(* Logix 5000 project; controller PRU vendor 1 type 14 code 107 rev 20.13; software revision 20.01; part 5 of 17 *)
(* tags used below, declared in another part *)
   AFI : BOOL;
   AlarmMaster : DINT;
   ALL_AUTO_IOK : BOOL;   // All equipment is in Auto Mode.
   ALL_DRIVES_ARE_CMD_FWD : BOOL;
   ALL_DRIVES_ARE_READY : BOOL;
   ALL_SHUTDOWN_FAULTS_IOK : BOOL;
   AUTO_DISCHARGE_CYCLE_ION : BOOL;   // Proces Sequencer (4-13)
   AUTO_SHUTDOWN_ENABLE : BOOL;
   CLEARING_PYROLIZER_TIME_REMAINING_SEC : REAL;
   CLEARING_PYROLIZER_TIME_REMAINING_TEMP : REAL;
   CLEARING_PYROLIZER_TIMER : TIMER;
   COOLSCREW : VFD;
   CR0_CON1_HTR1_GON : BOOL;   // ZONE 1 (L1,L2,L3)
   CR1_CON2_HTR2_GON : BOOL;   // ZONE 2 (L1,L2,L3)
   CR2_CON3_HTR3_GON : BOOL;   // ZONE 3 (L1,L2,L3)
   CR3_CON4_HTR4_GON : BOOL;   // ZONE 4 (L1) ZONE 5 (L2) ZONE 6 (L3)
   CR4_CON5_HTR5_GON : BOOL;   // ZONE 7 (L1) ZONE 8 (L2) ZONE 9 (L3)
   DRYER_MODE_AUTO : BOOL;
   FAULTS_FA1_IOK : BOOL;   // SYSTEM LEVEL FAULTS ARE OK.
   FAULTS_FA3A_IOK : BOOL;   // SCREWS DRIVES NOT FAULTED.
   FAULTS_FA3B_IOK : BOOL;   // ENCODERS NOT FAULTED.
   FAULTS_FA4_IOK : BOOL;   // HI TEMP FAULTS ARE OK.
   FAULTS_FA5_IOK : BOOL;
   FAULTS_FA5A_IOK : BOOL;   // COOLING SCREW FAULTS ARE OK.
   FAULTS_FA5C_IOK : BOOL;   // KG021 FAULTS ARE OK.
   FAULTS_FA5D_IOK : BOOL;   // KG021 FAULTS ARE OK.
   FAULTS_FA6_IOK : BOOL;   // HEATER FAULTS ARE OK.
   FINISH_PROCESS_TIME_REMAINING_SEC : REAL;
   FINISH_PROCESS_TIME_REMAINING_TEMP : REAL;
   FINISH_PROCESS_TIMER : TIMER;
   FS0101_ION : BOOL;   // LOW FLOW SWITCH - INLET AND DISCHARGE PURGE
   HEATER_FAULTS_IOK : BOOL;   // FA1, FA4, FA6
   HEATERS_CYCLE_ION : BOOL;   // Heaters are commanded on.
   HMI_ABORT_PB : BOOL;
   HMI_AUTO_START_PB : BOOL;
   HMI_CLEARING_PYROLIZER_TIME_MIN : REAL;
   HMI_FINISH_PROCESS_TIME_MIN : REAL;
   HMI_SHUTDOWN_PB : BOOL;
   HMI_SHUTDOWN_PURGE_TIME_MIN : REAL;
   HMI_STARTUP_PURGE_TIME_MIN : REAL;
   IFS_Status_Data : PLCStatusData;
   K0621_IS_OPEN : BOOL;
   K0622_IS_OPEN : BOOL;
   KG021_MODE : INT;   // 0 = OFF 1 = MAINT 2 = SEMI 3 = AUTO
   KG022_MODE : INT;   // 0 = OFF 1 = MAINT 2 = SEMI 3 = AUTO
   PID_ZONE_1 : PID;
   PID_ZONE_2 : PID;
   PID_ZONE_3 : PID;
   PID_ZONE_4 : PID;
   PID_ZONE_5 : PID;
   PID_ZONE_6 : PID;
   PID_ZONE_7 : PID;
   PID_ZONE_8 : PID;
   PID_ZONE_9 : PID;
   PROCESS_SEQUENCER : INT;
   PRODUCTION_ION : BOOL;
   SEQ_SHUTDOWN_ONS : BOOL;
   SEQ_STEP_00_DONE_TON : TIMER;
   SEQ_STEP_00_DONEA : BOOL;   // ALL_AUTO_IOK
   SEQ_STEP_00_DONEB : BOOL;   // ALL_DRIVES_ARE_READY
   SEQ_STEP_00_DONEC : BOOL;   // ALL_DRIVES_ARE_CMD_FWD
   SEQ_STEP_00_DONED : BOOL;   // ALL_SHUTDOWN_FAULTS_IOK
   SEQ_STEP_01_DONE_TON : TIMER;
   SEQ_STEP_01_DONEA : BOOL;   // FS-0204 INDICATES FLOW IS PRESENT
   SEQ_STEP_01_DONEB : BOOL;
   SEQ_STEP_01_DONEC : BOOL;
   SEQ_STEP_02_DONE_TON : TIMER;
   SEQ_STEP_02_DONEA : BOOL;   // FS-0101 INDICATES FLOW IS PRESENT
   SEQ_STEP_02_DONEB : BOOL;   // TIME > HMI SP (STARTUP PURGE)
   SEQ_STEP_02_DONEC : BOOL;
   SEQ_STEP_03_DONE_TON : TIMER;
   SEQ_STEP_03_DONEA : BOOL;   // HEATERS ARE ON.
   SEQ_STEP_03_DONEB : BOOL;
   SEQ_STEP_03_DONEC : BOOL;
   SEQ_STEP_04_DONE_TON : TIMER;
   SEQ_STEP_04_DONEA : BOOL;   // VFD0201 (ION)
   SEQ_STEP_04_DONEB : BOOL;   // KG-021 (OPEN 1X)
   SEQ_STEP_04_DONEC : BOOL;   // KF-022 (OPEN 1X)
   SEQ_STEP_05_DONE_TON : TIMER;
   SEQ_STEP_05_DONEA : BOOL;   // VFD0101 (ION)
   SEQ_STEP_05_DONEB : BOOL;   // VFD0102 (ION)
   SEQ_STEP_05_DONEC : BOOL;
   SEQ_STEP_06_DONE_TON : TIMER;
   SEQ_STEP_06_DONEA : BOOL;   // VFD0301 (ION)
   SEQ_STEP_06_DONEB : BOOL;
   SEQ_STEP_06_DONEC : BOOL;
   SEQ_STEP_07_DONE_TON : TIMER;
   SEQ_STEP_07_DONEA : BOOL;
   SEQ_STEP_07_DONEB : BOOL;
   SEQ_STEP_07_DONEC : BOOL;
   SEQ_STEP_07_DONED : BOOL;
   SEQ_STEP_08_DONE_TON : TIMER;
   SEQ_STEP_08_DONEA : BOOL;
   SEQ_STEP_08_DONEB : BOOL;
   SEQ_STEP_08_DONEC : BOOL;
   SEQ_STEP_09_DONE_TON : TIMER;
   SEQ_STEP_09_DONEA : BOOL;   // VFD0301 (IOF)
   SEQ_STEP_09_DONEB : BOOL;
   SEQ_STEP_09_DONEC : BOOL;
   SEQ_STEP_10_DONE_TON : TIMER;
   SEQ_STEP_10_DONEA : BOOL;   // TIME > HMI SP (FINISH PROCESS TIME)
   SEQ_STEP_10_DONEB : BOOL;
   SEQ_STEP_10_DONEC : BOOL;
   SEQ_STEP_11_DONE_TON : TIMER;
   SEQ_STEP_11_DONEA : BOOL;   // HEATERS ARE OFF.
   SEQ_STEP_11_DONEB : BOOL;
   SEQ_STEP_11_DONEC : BOOL;
   SEQ_STEP_12_DONE_TON : TIMER;
   SEQ_STEP_12_DONEA : BOOL;   // TIME > HMI SP (CLEARING TIME)
   SEQ_STEP_12_DONEB : BOOL;
   SEQ_STEP_12_DONEC : BOOL;
   SEQ_STEP_13_DONE_TON : TIMER;
   SEQ_STEP_13_DONEA : BOOL;   // VFD0101 (IOF)
   SEQ_STEP_13_DONEB : BOOL;   // VFD0102 (IOF)
   SEQ_STEP_13_DONEC : BOOL;
   SEQ_STEP_14_DONE_TON : TIMER;
   SEQ_STEP_14_DONEA : BOOL;   // VFD0201 (IOF)
   SEQ_STEP_14_DONEB : BOOL;   // KG-021 (CLOSED)
   SEQ_STEP_14_DONEC : BOOL;   // KF-022 (CLOSED)
   SEQ_STEP_15_DONE_TON : TIMER;
   SEQ_STEP_15_DONEA : BOOL;   // FS-0101 INDICATES FLOW IS PRESENT
   SEQ_STEP_15_DONEB : BOOL;   // TIME > HMI SP (SHUTDOWN PURGE)
   SEQ_STEP_15_DONEC : BOOL;
   SEQ_STEP_16_DONE_TON : TIMER;
   SEQ_STEP_16_DONEA : BOOL;   // ALL TEMPS < 200F
   SEQ_STEP_16_DONEB : BOOL;
   SEQ_STEP_16_DONEC : BOOL;
   SHUTDOWN_PURGE_TIME_REMAINING_SEC : REAL;
   SHUTDOWN_PURGE_TIME_REMAINING_TEMP : REAL;
   SHUTDOWN_PURGE_TIMER : TIMER;
   STANDBY_MODE_ION : BOOL;
   STANDBY_MODE_TON : TIMER;
   START_ENABLE : BOOL;
   STARTUP_PURGE_TIME_REMAINING_SEC : REAL;
   STARTUP_PURGE_TIME_REMAINING_TEMP : REAL;
   STARTUP_PURGE_TIMER : TIMER;
   STEP_00_ION : BOOL;   // 0 - SYSTEM NOT OPERATING
   STEP_01_ION : BOOL;   // 1 - COOLING WATER FLOW
   STEP_02_ION : BOOL;   // 2 - STARTUP N2 PURGE
   STEP_03_ION : BOOL;   // 3 - RAMPING HEATERS TO SETPOINT
   STEP_04_ION : BOOL;   // 4 - RUNNING DISCHARGE SYSTEM
   STEP_05_ION : BOOL;   // 5 - RUNNING PYROLIZER SCREWS
   STEP_06_ION : BOOL;   // 6 - RUNNING FEED SYSTEM
   STEP_07_ION : BOOL;   // 7 - SYSTEM PROCESSING
   STEP_08_ION : BOOL;   // 8 - AUTO SHUTDOWN
   STEP_09_ION : BOOL;   // 9 - STOPPING FEED SYSTEM
   STEP_10_ION : BOOL;   // 10 - FINISHING PROCESS
   STEP_11_ION : BOOL;   // 11 - STOPPING HEATERS
   STEP_12_ION : BOOL;   // 12 - CLEARING PYROLIZER
   STEP_13_ION : BOOL;   // 13 - STOPPING PYROLIZER
   STEP_14_ION : BOOL;   // 14 - STOPPING DISCHARGE SYSTEM
   STEP_15_ION : BOOL;   // 15 - SHUTDOWN N2 PURGE
   STEP_16_ION : BOOL;   // 16 - WAITING FOR SYSTEM COOL
   TE0101 : REAL;
   TE0102 : REAL;
   TE0103 : REAL;
   TE0104 : REAL;
   TE0105 : REAL;
   TE0106 : REAL;
   TE0107 : REAL;
   TE0108 : REAL;
   TE0109 : REAL;
   TE0110 : REAL;
   TE0111 : REAL;
   TE0112 : REAL;
   TE0113 : REAL;
   TE0114 : REAL;
   TE0115 : REAL;
   TE0116 : REAL;
   TE0117 : REAL;
   TE0118 : REAL;
   TE0119 : REAL;
   TE0120 : REAL;
   TE0121 : REAL;
   TE0122 : REAL;
   TE0123 : REAL;
   TE0124 : REAL;
   TE0125 : REAL;
   TE0126 : REAL;
   TE0127 : REAL;
   TE0128 : REAL;
   TE0129 : REAL;
   TE0130 : REAL;
   TE0201 : REAL;
   TE0202 : REAL;
   TOTE_CHANGE_TIMED_OUT : BOOL;
   UTL_CommsLossAlm : BOOL;   // Comms to UTL Has been Lost Alarm
   UTL_CommsWarningAlm : BOOL;   // Comms to UTL Has been Lost Warning Alarm
   UTL_Status_Data : PLCStatusData;
   WARNA_IOK : BOOL;
   WARNB_IOK : BOOL;
   WARNC_IOK : BOOL;
   WARND_IOK : BOOL;
   WARNE_IOK : BOOL;
   WARNF_IOK : BOOL;
   WARNG_IOK : BOOL;
   WARNING_FAULTS_IOK : BOOL;
(* MainProgram, continued *)

ROUTINE A11_SEQUENCER_PROCESS   (* ladder *)
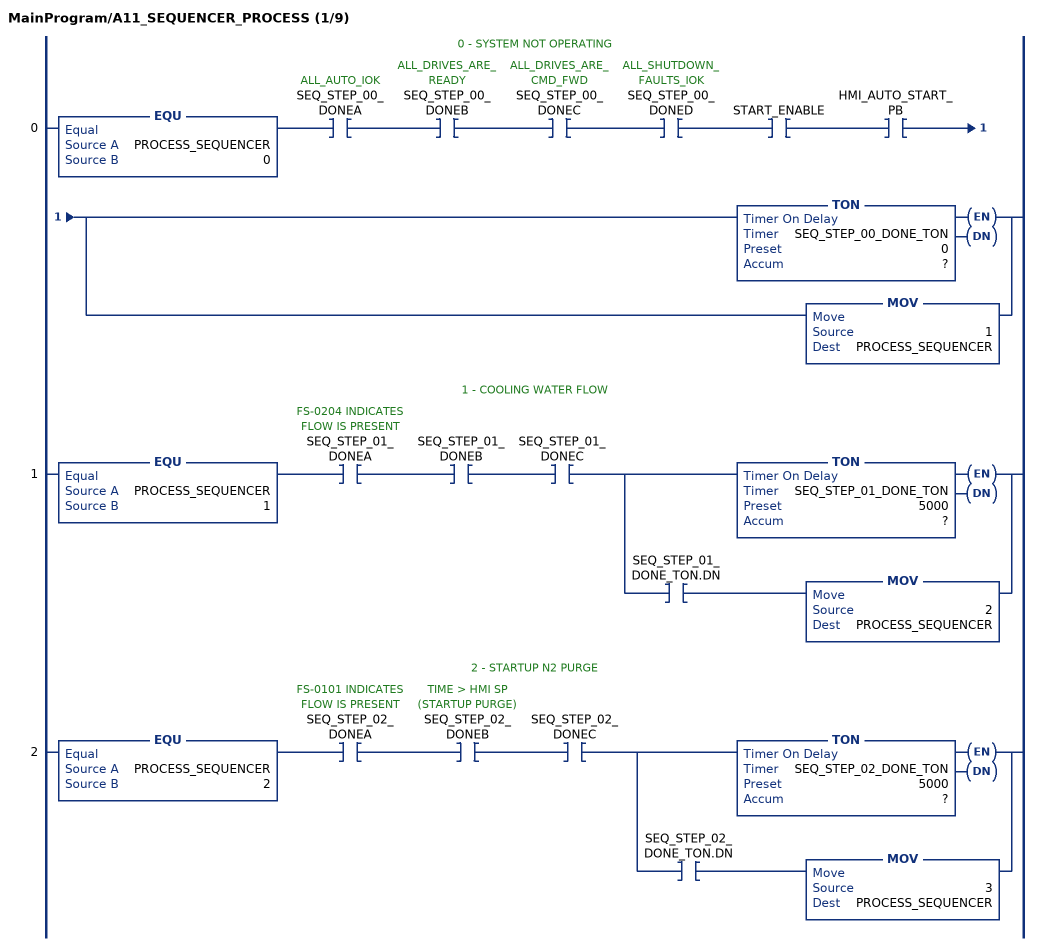
   // 0 - SYSTEM NOT OPERATING
   0: EQU(PROCESS_SEQUENCER,0)XIC(SEQ_STEP_00_DONEA)XIC(SEQ_STEP_00_DONEB)XIC(SEQ_STEP_00_DONEC)XIC(SEQ_STEP_00_DONED)XIC(START_ENABLE)XIC(HMI_AUTO_START_PB)[TON(SEQ_STEP_00_DONE_TON,?,?) ,MOV(1,PROCESS_SEQUENCER) ];
   // 1 - COOLING WATER FLOW
   1: EQU(PROCESS_SEQUENCER,1)XIC(SEQ_STEP_01_DONEA)XIC(SEQ_STEP_01_DONEB)XIC(SEQ_STEP_01_DONEC)[TON(SEQ_STEP_01_DONE_TON,?,?) ,XIC(SEQ_STEP_01_DONE_TON.DN) MOV(2,PROCESS_SEQUENCER) ];
   // 2 - STARTUP N2 PURGE
   2: EQU(PROCESS_SEQUENCER,2)XIC(SEQ_STEP_02_DONEA)XIC(SEQ_STEP_02_DONEB)XIC(SEQ_STEP_02_DONEC)[TON(SEQ_STEP_02_DONE_TON,?,?) ,XIC(SEQ_STEP_02_DONE_TON.DN) MOV(3,PROCESS_SEQUENCER) ];
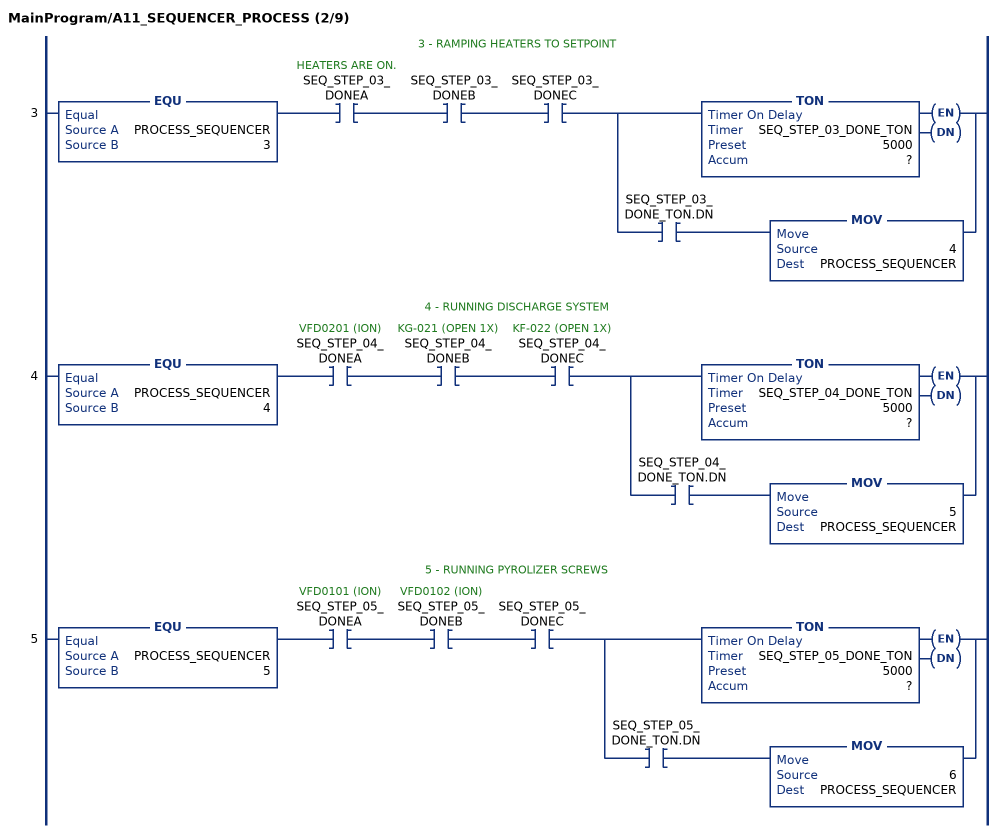
   // 3 - RAMPING HEATERS TO SETPOINT
   3: EQU(PROCESS_SEQUENCER,3)XIC(SEQ_STEP_03_DONEA)XIC(SEQ_STEP_03_DONEB)XIC(SEQ_STEP_03_DONEC)[TON(SEQ_STEP_03_DONE_TON,?,?) ,XIC(SEQ_STEP_03_DONE_TON.DN) MOV(4,PROCESS_SEQUENCER) ];
   // 4 - RUNNING DISCHARGE SYSTEM
   4: EQU(PROCESS_SEQUENCER,4)XIC(SEQ_STEP_04_DONEA)XIC(SEQ_STEP_04_DONEB)XIC(SEQ_STEP_04_DONEC)[TON(SEQ_STEP_04_DONE_TON,?,?) ,XIC(SEQ_STEP_04_DONE_TON.DN) MOV(5,PROCESS_SEQUENCER) ];
   // 5 - RUNNING PYROLIZER SCREWS
   5: EQU(PROCESS_SEQUENCER,5)XIC(SEQ_STEP_05_DONEA)XIC(SEQ_STEP_05_DONEB)XIC(SEQ_STEP_05_DONEC)[TON(SEQ_STEP_05_DONE_TON,?,?) ,XIC(SEQ_STEP_05_DONE_TON.DN) MOV(6,PROCESS_SEQUENCER) ];
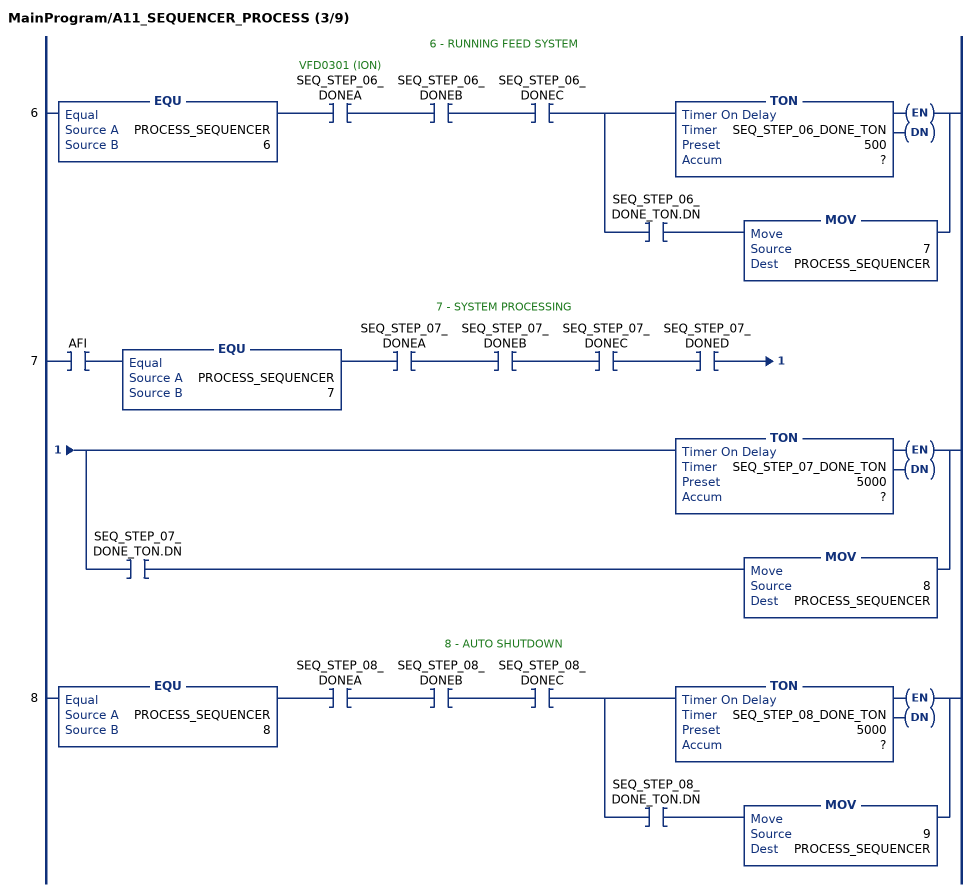
   // 6 - RUNNING FEED SYSTEM
   6: EQU(PROCESS_SEQUENCER,6)XIC(SEQ_STEP_06_DONEA)XIC(SEQ_STEP_06_DONEB)XIC(SEQ_STEP_06_DONEC)[TON(SEQ_STEP_06_DONE_TON,?,?) ,XIC(SEQ_STEP_06_DONE_TON.DN) MOV(7,PROCESS_SEQUENCER) ];
   // 7 - SYSTEM PROCESSING
   7: XIC(AFI)EQU(PROCESS_SEQUENCER,7)XIC(SEQ_STEP_07_DONEA)XIC(SEQ_STEP_07_DONEB)XIC(SEQ_STEP_07_DONEC)XIC(SEQ_STEP_07_DONED)[TON(SEQ_STEP_07_DONE_TON,?,?) ,XIC(SEQ_STEP_07_DONE_TON.DN) MOV(8,PROCESS_SEQUENCER) ];
   // 8 - AUTO SHUTDOWN
   8: EQU(PROCESS_SEQUENCER,8)XIC(SEQ_STEP_08_DONEA)XIC(SEQ_STEP_08_DONEB)XIC(SEQ_STEP_08_DONEC)[TON(SEQ_STEP_08_DONE_TON,?,?) ,XIC(SEQ_STEP_08_DONE_TON.DN) MOV(9,PROCESS_SEQUENCER) ];
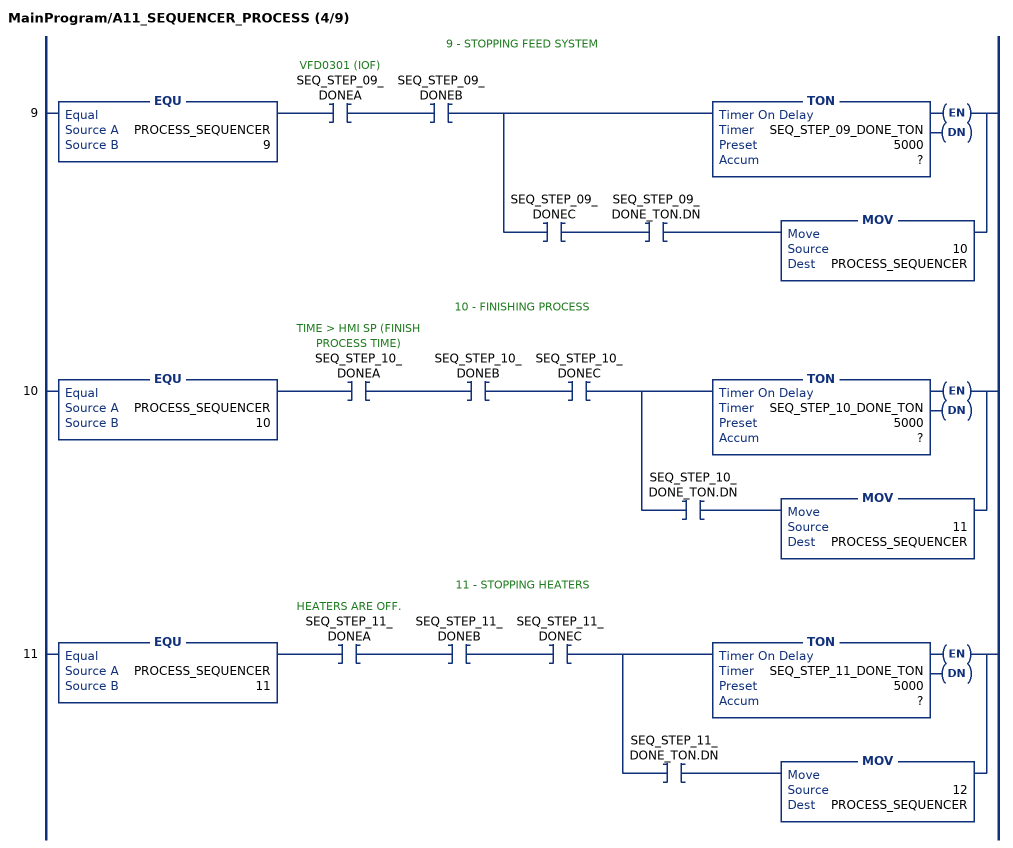
   // 9 - STOPPING FEED SYSTEM
   9: EQU(PROCESS_SEQUENCER,9)XIC(SEQ_STEP_09_DONEA)XIC(SEQ_STEP_09_DONEB)[TON(SEQ_STEP_09_DONE_TON,?,?) ,XIC(SEQ_STEP_09_DONEC) XIC(SEQ_STEP_09_DONE_TON.DN) MOV(10,PROCESS_SEQUENCER) ];
   // 10 - FINISHING PROCESS
   10: EQU(PROCESS_SEQUENCER,10)XIC(SEQ_STEP_10_DONEA)XIC(SEQ_STEP_10_DONEB)XIC(SEQ_STEP_10_DONEC)[TON(SEQ_STEP_10_DONE_TON,?,?) ,XIC(SEQ_STEP_10_DONE_TON.DN) MOV(11,PROCESS_SEQUENCER) ];
   // 11 - STOPPING HEATERS
   11: EQU(PROCESS_SEQUENCER,11)XIC(SEQ_STEP_11_DONEA)XIC(SEQ_STEP_11_DONEB)XIC(SEQ_STEP_11_DONEC)[TON(SEQ_STEP_11_DONE_TON,?,?) ,XIC(SEQ_STEP_11_DONE_TON.DN) MOV(12,PROCESS_SEQUENCER) ];
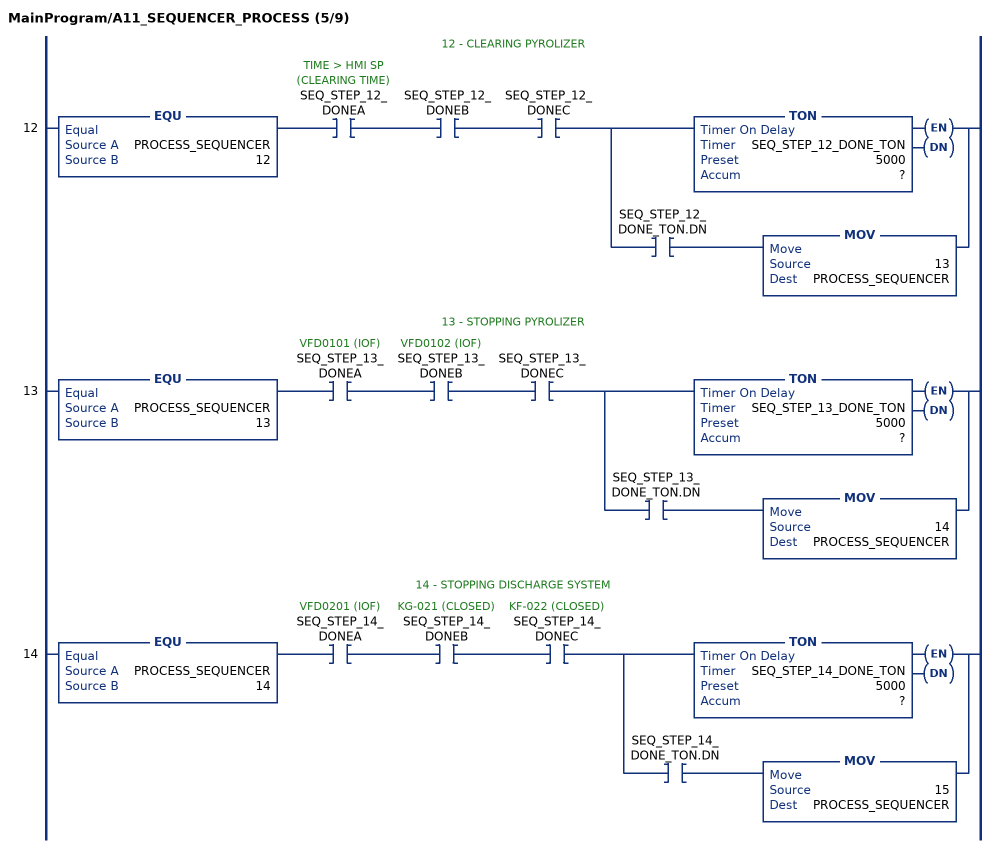
   // 12 - CLEARING PYROLIZER
   12: EQU(PROCESS_SEQUENCER,12)XIC(SEQ_STEP_12_DONEA)XIC(SEQ_STEP_12_DONEB)XIC(SEQ_STEP_12_DONEC)[TON(SEQ_STEP_12_DONE_TON,?,?) ,XIC(SEQ_STEP_12_DONE_TON.DN) MOV(13,PROCESS_SEQUENCER) ];
   // 13 - STOPPING PYROLIZER
   13: EQU(PROCESS_SEQUENCER,13)XIC(SEQ_STEP_13_DONEA)XIC(SEQ_STEP_13_DONEB)XIC(SEQ_STEP_13_DONEC)[TON(SEQ_STEP_13_DONE_TON,?,?) ,XIC(SEQ_STEP_13_DONE_TON.DN) MOV(14,PROCESS_SEQUENCER) ];
   // 14 - STOPPING DISCHARGE SYSTEM
   14: EQU(PROCESS_SEQUENCER,14)XIC(SEQ_STEP_14_DONEA)XIC(SEQ_STEP_14_DONEB)XIC(SEQ_STEP_14_DONEC)[TON(SEQ_STEP_14_DONE_TON,?,?) ,XIC(SEQ_STEP_14_DONE_TON.DN) MOV(15,PROCESS_SEQUENCER) ];
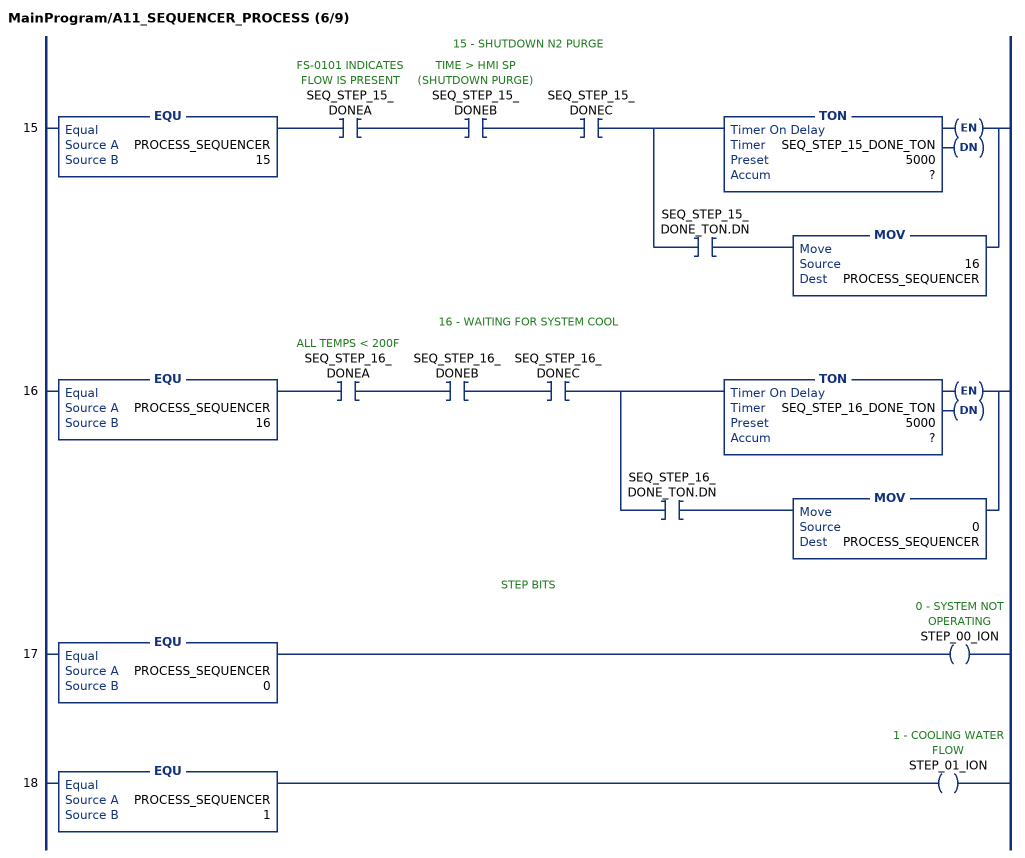
   // 15 - SHUTDOWN N2 PURGE
   15: EQU(PROCESS_SEQUENCER,15)XIC(SEQ_STEP_15_DONEA)XIC(SEQ_STEP_15_DONEB)XIC(SEQ_STEP_15_DONEC)[TON(SEQ_STEP_15_DONE_TON,?,?) ,XIC(SEQ_STEP_15_DONE_TON.DN) MOV(16,PROCESS_SEQUENCER) ];
   // 16 - WAITING FOR SYSTEM COOL
   16: EQU(PROCESS_SEQUENCER,16)XIC(SEQ_STEP_16_DONEA)XIC(SEQ_STEP_16_DONEB)XIC(SEQ_STEP_16_DONEC)[TON(SEQ_STEP_16_DONE_TON,?,?) ,XIC(SEQ_STEP_16_DONE_TON.DN) MOV(0,PROCESS_SEQUENCER) ];
   // STEP BITS
   17: EQU(PROCESS_SEQUENCER,0)OTE(STEP_00_ION);
   18: EQU(PROCESS_SEQUENCER,1)OTE(STEP_01_ION);
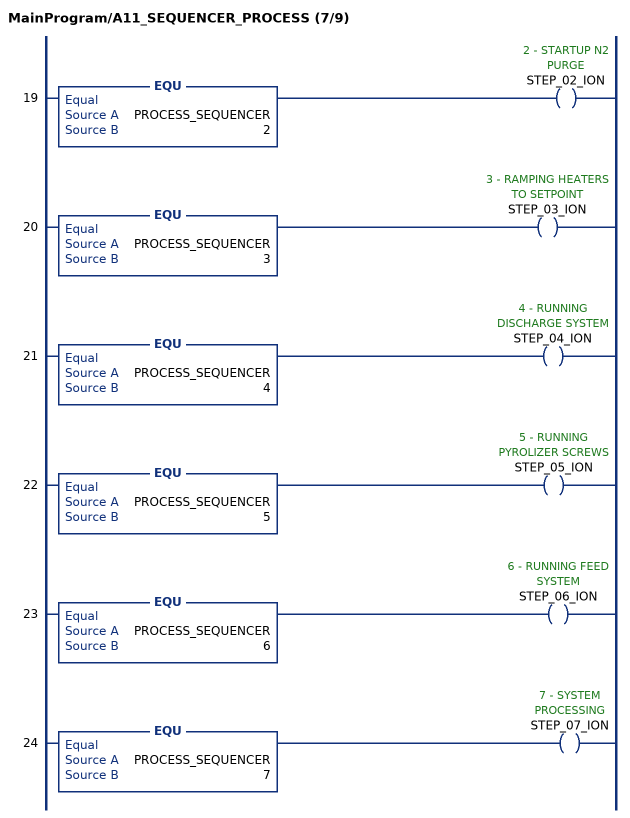
   19: EQU(PROCESS_SEQUENCER,2)OTE(STEP_02_ION);
   20: EQU(PROCESS_SEQUENCER,3)OTE(STEP_03_ION);
   21: EQU(PROCESS_SEQUENCER,4)OTE(STEP_04_ION);
   22: EQU(PROCESS_SEQUENCER,5)OTE(STEP_05_ION);
   23: EQU(PROCESS_SEQUENCER,6)OTE(STEP_06_ION);
   24: EQU(PROCESS_SEQUENCER,7)OTE(STEP_07_ION);
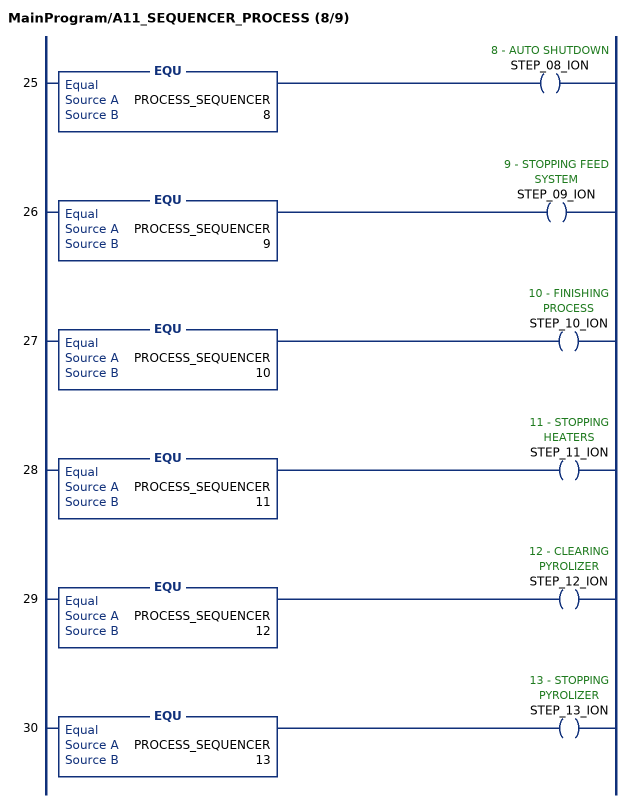
   25: EQU(PROCESS_SEQUENCER,8)OTE(STEP_08_ION);
   26: EQU(PROCESS_SEQUENCER,9)OTE(STEP_09_ION);
   27: EQU(PROCESS_SEQUENCER,10)OTE(STEP_10_ION);
   28: EQU(PROCESS_SEQUENCER,11)OTE(STEP_11_ION);
   29: EQU(PROCESS_SEQUENCER,12)OTE(STEP_12_ION);
   30: EQU(PROCESS_SEQUENCER,13)OTE(STEP_13_ION);
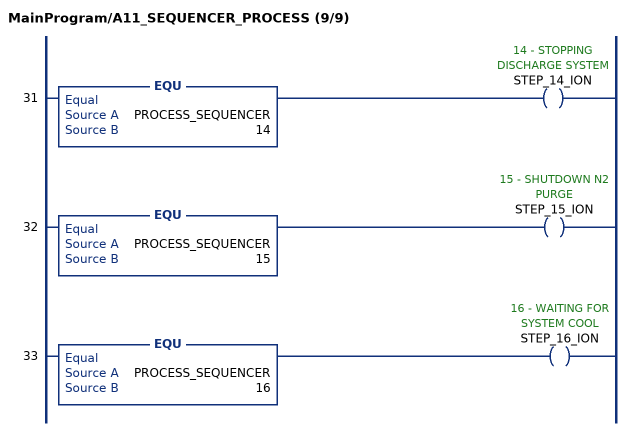
   31: EQU(PROCESS_SEQUENCER,14)OTE(STEP_14_ION);
   32: EQU(PROCESS_SEQUENCER,15)OTE(STEP_15_ION);
   33: EQU(PROCESS_SEQUENCER,16)OTE(STEP_16_ION);
END_ROUTINE

ROUTINE A12_SEQ_PROCESS_Permissives   (* ladder *)
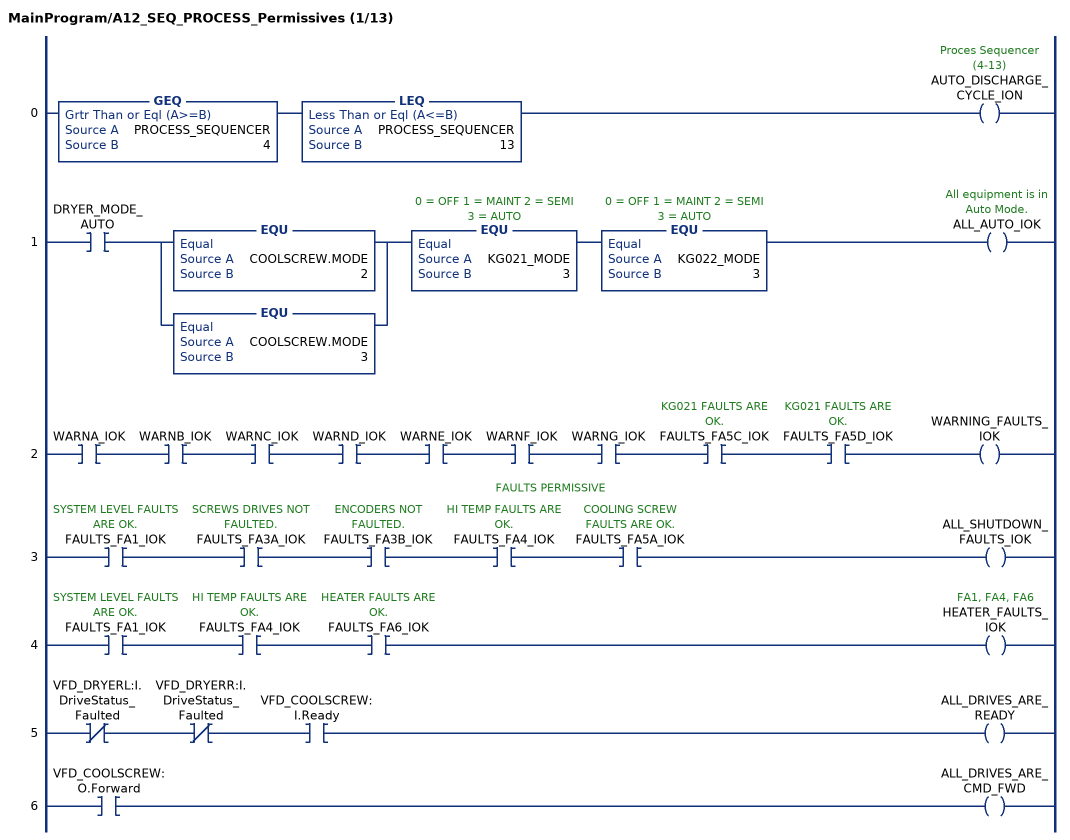
   0: GEQ(PROCESS_SEQUENCER,4)LEQ(PROCESS_SEQUENCER,13)OTE(AUTO_DISCHARGE_CYCLE_ION);
   1: XIC(DRYER_MODE_AUTO)[EQU(COOLSCREW.MODE,2) ,EQU(COOLSCREW.MODE,3) ]EQU(KG021_MODE,3)EQU(KG022_MODE,3)OTE(ALL_AUTO_IOK);
   2: XIC(WARNA_IOK)XIC(WARNB_IOK)XIC(WARNC_IOK)XIC(WARND_IOK)XIC(WARNE_IOK)XIC(WARNF_IOK)XIC(WARNG_IOK)XIC(FAULTS_FA5C_IOK)XIC(FAULTS_FA5D_IOK)OTE(WARNING_FAULTS_IOK);
   // FAULTS PERMISSIVE
   3: XIC(FAULTS_FA1_IOK)XIC(FAULTS_FA3A_IOK)XIC(FAULTS_FA3B_IOK)XIC(FAULTS_FA4_IOK)XIC(FAULTS_FA5A_IOK)OTE(ALL_SHUTDOWN_FAULTS_IOK);
   4: XIC(FAULTS_FA1_IOK)XIC(FAULTS_FA4_IOK)XIC(FAULTS_FA6_IOK)OTE(HEATER_FAULTS_IOK);
   5: XIO(VFD_DRYERL:I.DriveStatus_Faulted)XIO(VFD_DRYERR:I.DriveStatus_Faulted)XIC(VFD_COOLSCREW:I.Ready)OTE(ALL_DRIVES_ARE_READY);
   6: XIC(VFD_COOLSCREW:O.Forward)OTE(ALL_DRIVES_ARE_CMD_FWD);
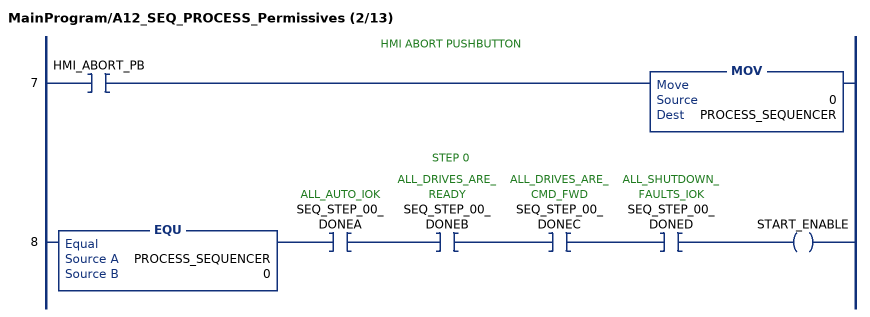
   // HMI ABORT PUSHBUTTON
   7: XIC(HMI_ABORT_PB)MOV(0,PROCESS_SEQUENCER);
   // STEP 0
   8: EQU(PROCESS_SEQUENCER,0)XIC(SEQ_STEP_00_DONEA)XIC(SEQ_STEP_00_DONEB)XIC(SEQ_STEP_00_DONEC)XIC(SEQ_STEP_00_DONED)OTE(START_ENABLE);
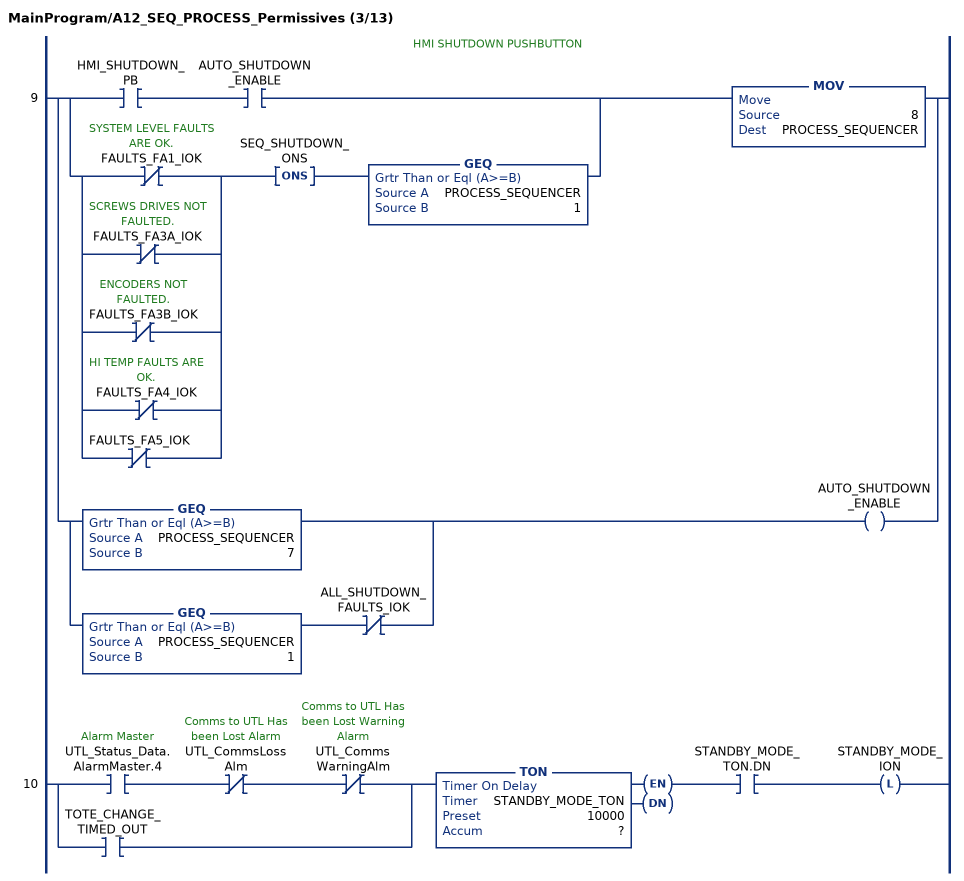
   // HMI SHUTDOWN PUSHBUTTON
   9: [[XIC(HMI_SHUTDOWN_PB) XIC(AUTO_SHUTDOWN_ENABLE) ,[XIO(FAULTS_FA1_IOK) ,XIO(FAULTS_FA3A_IOK) ,XIO(FAULTS_FA3B_IOK) ,XIO(FAULTS_FA4_IOK) ,XIO(FAULTS_FA5_IOK) ] ONS(SEQ_SHUTDOWN_ONS) GEQ(PROCESS_SEQUENCER,1) ] MOV(8,PROCESS_SEQUENCER) ,[GEQ(PROCESS_SEQUENCER,7) ,GEQ(PROCESS_SEQUENCER,1) XIO(ALL_SHUTDOWN_FAULTS_IOK) ] OTE(AUTO_SHUTDOWN_ENABLE) ];
   10: [XIC(UTL_Status_Data.AlarmMaster.4) XIO(UTL_CommsLossAlm) XIO(UTL_CommsWarningAlm) ,XIC(TOTE_CHANGE_TIMED_OUT) ]TON(STANDBY_MODE_TON,?,?)XIC(STANDBY_MODE_TON.DN)OTL(STANDBY_MODE_ION);
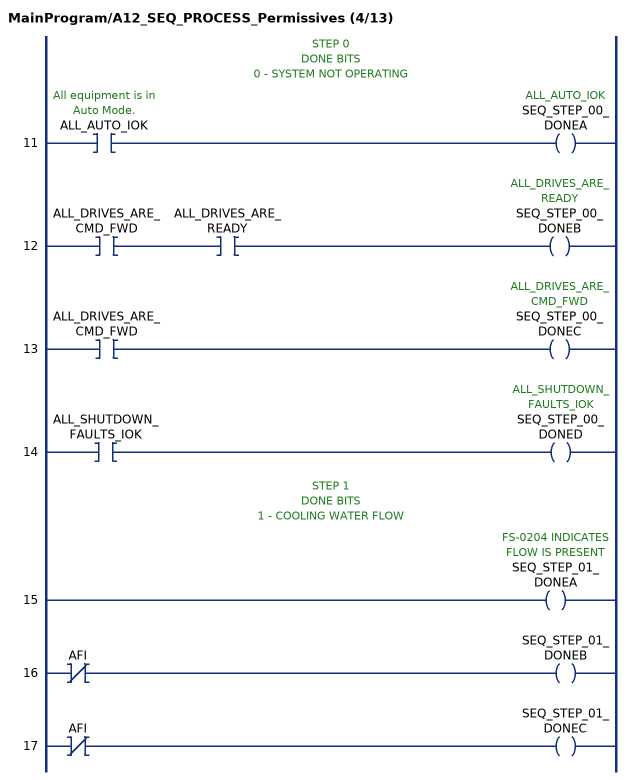
   // STEP 0
   // DONE BITS
   // 0 - SYSTEM NOT OPERATING
   11: XIC(ALL_AUTO_IOK)OTE(SEQ_STEP_00_DONEA);
   12: XIC(ALL_DRIVES_ARE_CMD_FWD)XIC(ALL_DRIVES_ARE_READY)OTE(SEQ_STEP_00_DONEB);
   13: XIC(ALL_DRIVES_ARE_CMD_FWD)OTE(SEQ_STEP_00_DONEC);
   14: XIC(ALL_SHUTDOWN_FAULTS_IOK)OTE(SEQ_STEP_00_DONED);
   // STEP 1
   // DONE BITS
   // 1 - COOLING WATER FLOW
   15: OTE(SEQ_STEP_01_DONEA);
   16: XIO(AFI)OTE(SEQ_STEP_01_DONEB);
   17: XIO(AFI)OTE(SEQ_STEP_01_DONEC);
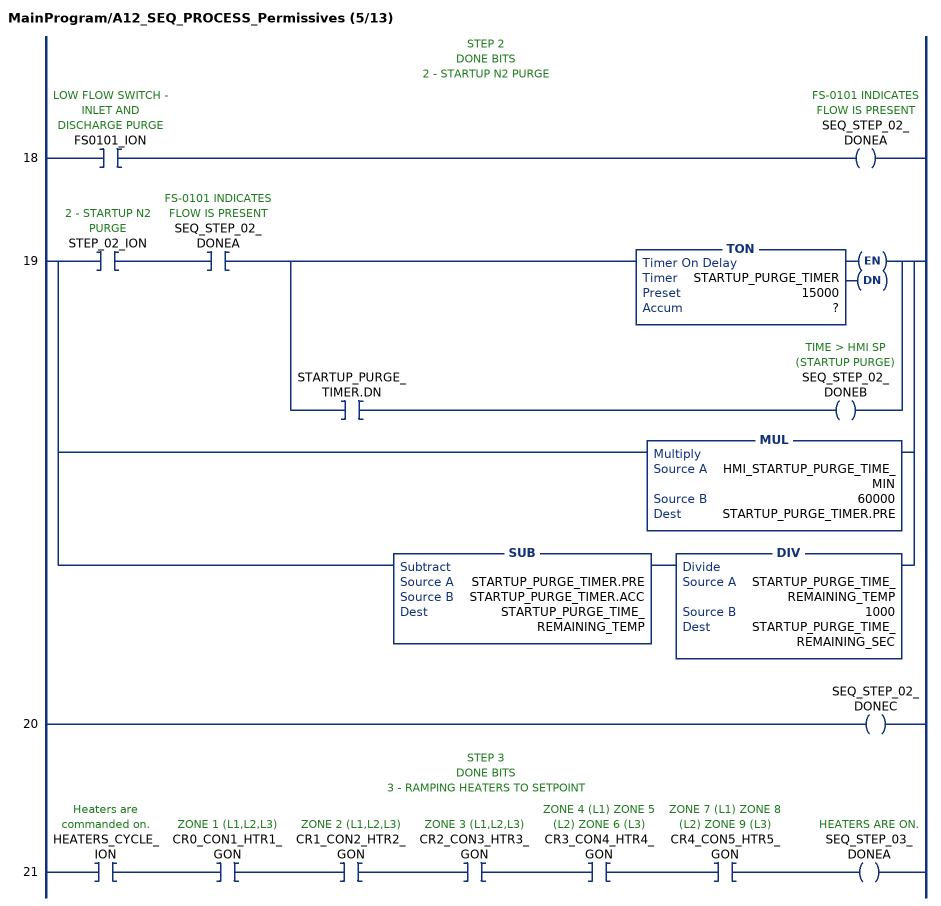
   // STEP 2
   // DONE BITS
   // 2 - STARTUP N2 PURGE
   18: XIC(FS0101_ION)OTE(SEQ_STEP_02_DONEA);
   19: [XIC(STEP_02_ION) XIC(SEQ_STEP_02_DONEA) [TON(STARTUP_PURGE_TIMER,?,?) ,XIC(STARTUP_PURGE_TIMER.DN) OTE(SEQ_STEP_02_DONEB) ] ,MUL(HMI_STARTUP_PURGE_TIME_MIN,60000,STARTUP_PURGE_TIMER.PRE) ,SUB(STARTUP_PURGE_TIMER.PRE,STARTUP_PURGE_TIMER.ACC,STARTUP_PURGE_TIME_REMAINING_TEMP) DIV(STARTUP_PURGE_TIME_REMAINING_TEMP,1000,STARTUP_PURGE_TIME_REMAINING_SEC) ];
   20: OTE(SEQ_STEP_02_DONEC);
   // STEP 3
   // DONE BITS
   // 3 - RAMPING HEATERS TO SETPOINT
   21: XIC(HEATERS_CYCLE_ION)XIC(CR0_CON1_HTR1_GON)XIC(CR1_CON2_HTR2_GON)XIC(CR2_CON3_HTR3_GON)XIC(CR3_CON4_HTR4_GON)XIC(CR4_CON5_HTR5_GON)OTE(SEQ_STEP_03_DONEA);
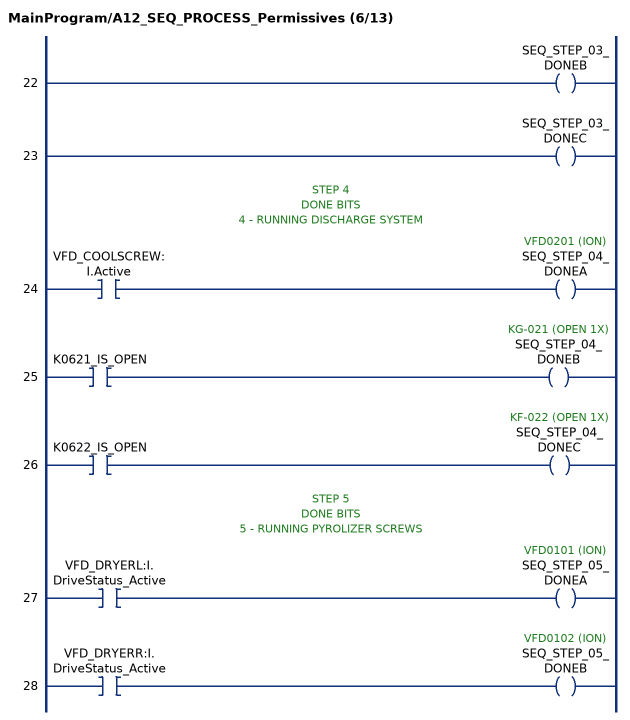
   22: OTE(SEQ_STEP_03_DONEB);
   23: OTE(SEQ_STEP_03_DONEC);
   // STEP 4
   // DONE BITS
   // 4 - RUNNING DISCHARGE SYSTEM
   24: XIC(VFD_COOLSCREW:I.Active)OTE(SEQ_STEP_04_DONEA);
   25: XIC(K0621_IS_OPEN)OTE(SEQ_STEP_04_DONEB);
   26: XIC(K0622_IS_OPEN)OTE(SEQ_STEP_04_DONEC);
   // STEP 5
   // DONE BITS
   // 5 - RUNNING PYROLIZER SCREWS
   27: XIC(VFD_DRYERL:I.DriveStatus_Active)OTE(SEQ_STEP_05_DONEA);
   28: XIC(VFD_DRYERR:I.DriveStatus_Active)OTE(SEQ_STEP_05_DONEB);
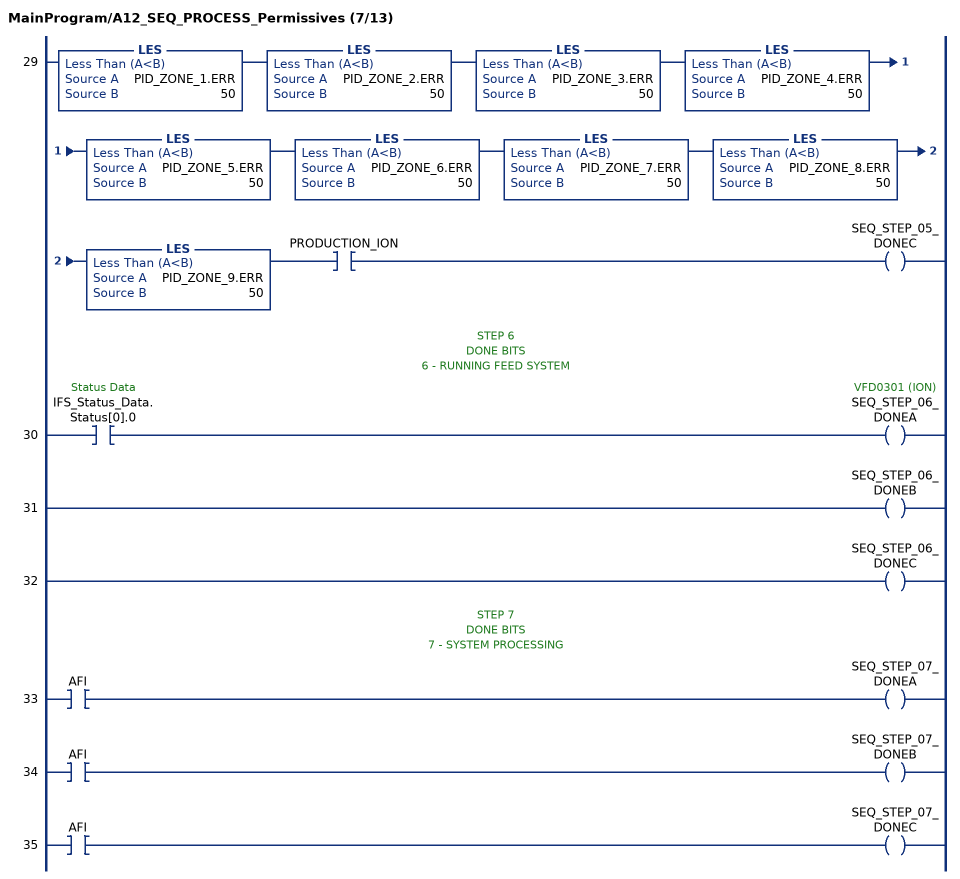
   29: LES(PID_ZONE_1.ERR,50)LES(PID_ZONE_2.ERR,50)LES(PID_ZONE_3.ERR,50)LES(PID_ZONE_4.ERR,50)LES(PID_ZONE_5.ERR,50)LES(PID_ZONE_6.ERR,50)LES(PID_ZONE_7.ERR,50)LES(PID_ZONE_8.ERR,50)LES(PID_ZONE_9.ERR,50)XIC(PRODUCTION_ION)OTE(SEQ_STEP_05_DONEC);
   // STEP 6
   // DONE BITS
   // 6 - RUNNING FEED SYSTEM
   30: XIC(IFS_Status_Data.Status[0].0)OTE(SEQ_STEP_06_DONEA);
   31: OTE(SEQ_STEP_06_DONEB);
   32: OTE(SEQ_STEP_06_DONEC);
   // STEP 7
   // DONE BITS
   // 7 - SYSTEM PROCESSING
   33: XIC(AFI)OTE(SEQ_STEP_07_DONEA);
   34: XIC(AFI)OTE(SEQ_STEP_07_DONEB);
   35: XIC(AFI)OTE(SEQ_STEP_07_DONEC);
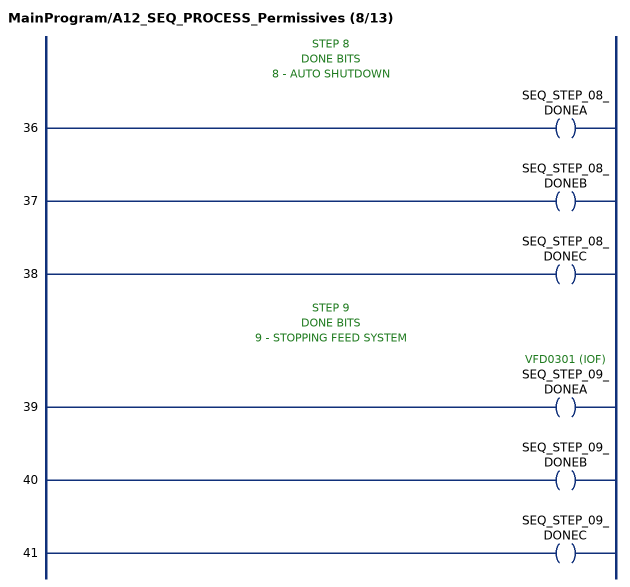
   // STEP 8
   // DONE BITS
   // 8 - AUTO SHUTDOWN
   36: OTE(SEQ_STEP_08_DONEA);
   37: OTE(SEQ_STEP_08_DONEB);
   38: OTE(SEQ_STEP_08_DONEC);
   // STEP 9
   // DONE BITS
   // 9 - STOPPING FEED SYSTEM
   39: OTE(SEQ_STEP_09_DONEA);
   40: OTE(SEQ_STEP_09_DONEB);
   41: OTE(SEQ_STEP_09_DONEC);
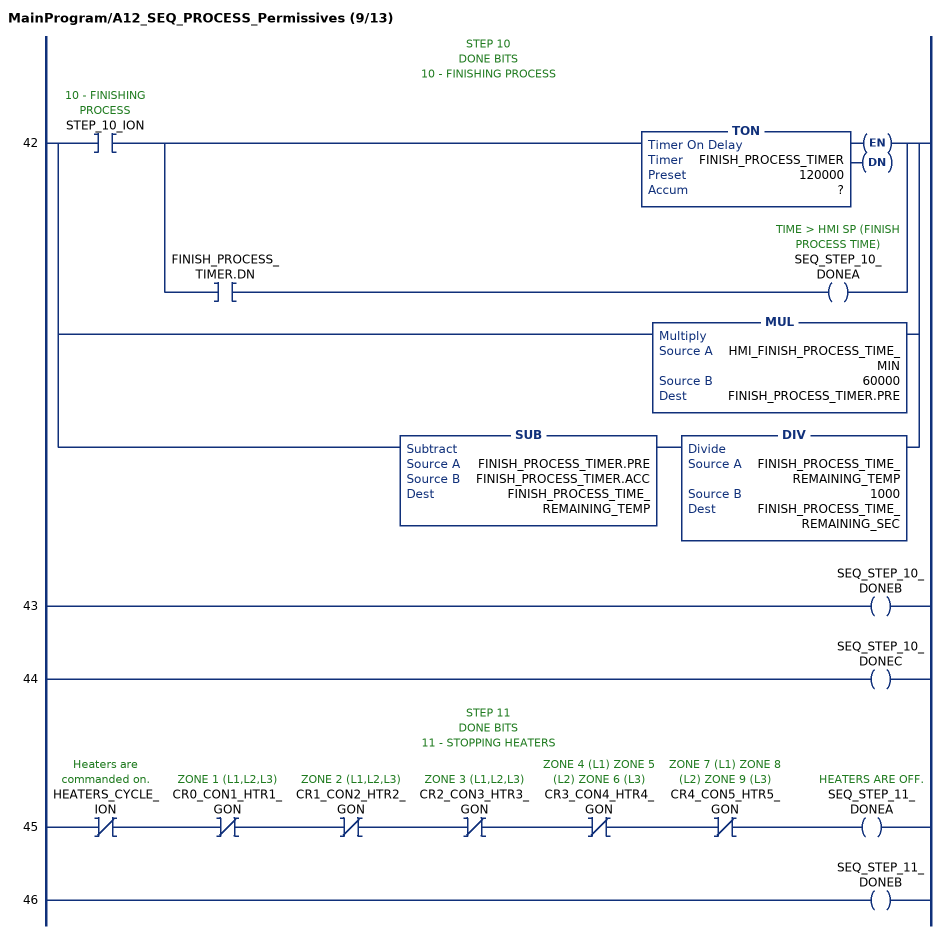
   // STEP 10
   // DONE BITS
   // 10 - FINISHING PROCESS
   42: [XIC(STEP_10_ION) [TON(FINISH_PROCESS_TIMER,?,?) ,XIC(FINISH_PROCESS_TIMER.DN) OTE(SEQ_STEP_10_DONEA) ] ,MUL(HMI_FINISH_PROCESS_TIME_MIN,60000,FINISH_PROCESS_TIMER.PRE) ,SUB(FINISH_PROCESS_TIMER.PRE,FINISH_PROCESS_TIMER.ACC,FINISH_PROCESS_TIME_REMAINING_TEMP) DIV(FINISH_PROCESS_TIME_REMAINING_TEMP,1000,FINISH_PROCESS_TIME_REMAINING_SEC) ];
   43: OTE(SEQ_STEP_10_DONEB);
   44: OTE(SEQ_STEP_10_DONEC);
   // STEP 11
   // DONE BITS
   // 11 - STOPPING HEATERS
   45: XIO(HEATERS_CYCLE_ION)XIO(CR0_CON1_HTR1_GON)XIO(CR1_CON2_HTR2_GON)XIO(CR2_CON3_HTR3_GON)XIO(CR3_CON4_HTR4_GON)XIO(CR4_CON5_HTR5_GON)OTE(SEQ_STEP_11_DONEA);
   46: OTE(SEQ_STEP_11_DONEB);
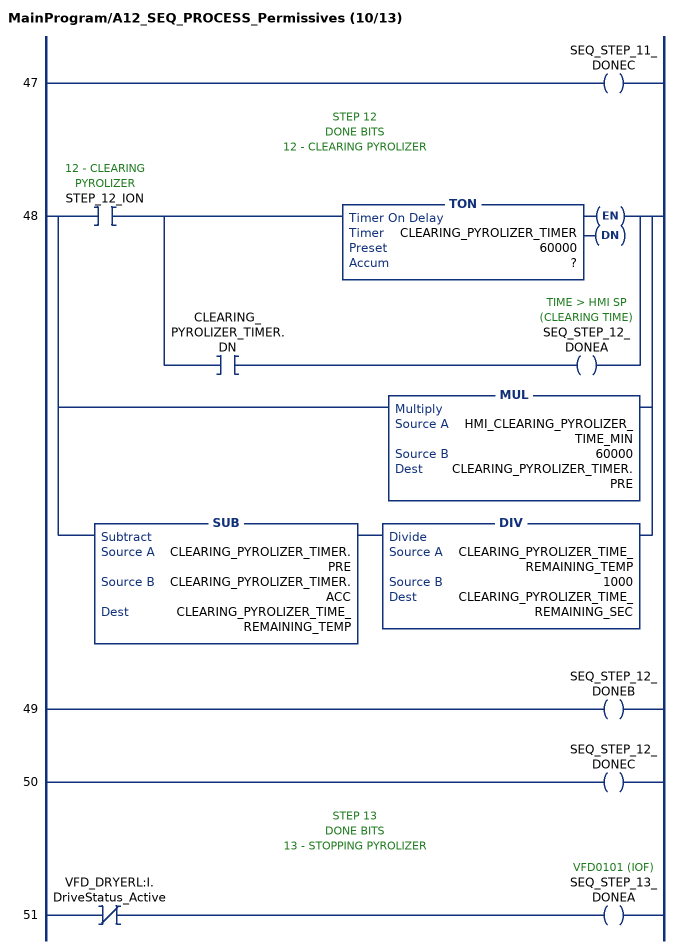
   47: OTE(SEQ_STEP_11_DONEC);
   // STEP 12
   // DONE BITS
   // 12 - CLEARING PYROLIZER
   48: [XIC(STEP_12_ION) [TON(CLEARING_PYROLIZER_TIMER,?,?) ,XIC(CLEARING_PYROLIZER_TIMER.DN) OTE(SEQ_STEP_12_DONEA) ] ,MUL(HMI_CLEARING_PYROLIZER_TIME_MIN,60000,CLEARING_PYROLIZER_TIMER.PRE) ,SUB(CLEARING_PYROLIZER_TIMER.PRE,CLEARING_PYROLIZER_TIMER.ACC,CLEARING_PYROLIZER_TIME_REMAINING_TEMP) DIV(CLEARING_PYROLIZER_TIME_REMAINING_TEMP,1000,CLEARING_PYROLIZER_TIME_REMAINING_SEC) ];
   49: OTE(SEQ_STEP_12_DONEB);
   50: OTE(SEQ_STEP_12_DONEC);
   // STEP 13
   // DONE BITS
   // 13 - STOPPING PYROLIZER
   51: XIO(VFD_DRYERL:I.DriveStatus_Active)OTE(SEQ_STEP_13_DONEA);
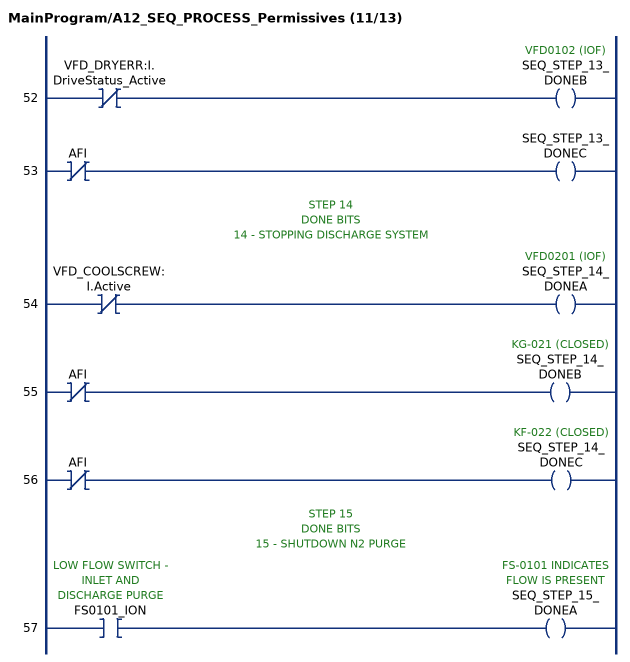
   52: XIO(VFD_DRYERR:I.DriveStatus_Active)OTE(SEQ_STEP_13_DONEB);
   53: XIO(AFI)OTE(SEQ_STEP_13_DONEC);
   // STEP 14
   // DONE BITS
   // 14 - STOPPING DISCHARGE SYSTEM
   54: XIO(VFD_COOLSCREW:I.Active)OTE(SEQ_STEP_14_DONEA);
   55: XIO(AFI)OTE(SEQ_STEP_14_DONEB);
   56: XIO(AFI)OTE(SEQ_STEP_14_DONEC);
   // STEP 15
   // DONE BITS
   // 15 - SHUTDOWN N2 PURGE
   57: XIC(FS0101_ION)OTE(SEQ_STEP_15_DONEA);
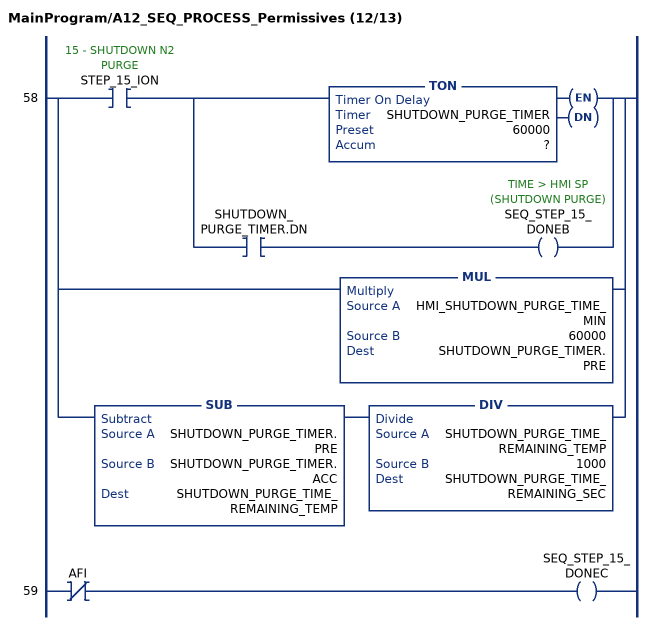
   58: [XIC(STEP_15_ION) [TON(SHUTDOWN_PURGE_TIMER,?,?) ,XIC(SHUTDOWN_PURGE_TIMER.DN) OTE(SEQ_STEP_15_DONEB) ] ,MUL(HMI_SHUTDOWN_PURGE_TIME_MIN,60000,SHUTDOWN_PURGE_TIMER.PRE) ,SUB(SHUTDOWN_PURGE_TIMER.PRE,SHUTDOWN_PURGE_TIMER.ACC,SHUTDOWN_PURGE_TIME_REMAINING_TEMP) DIV(SHUTDOWN_PURGE_TIME_REMAINING_TEMP,1000,SHUTDOWN_PURGE_TIME_REMAINING_SEC) ];
   59: XIO(AFI)OTE(SEQ_STEP_15_DONEC);
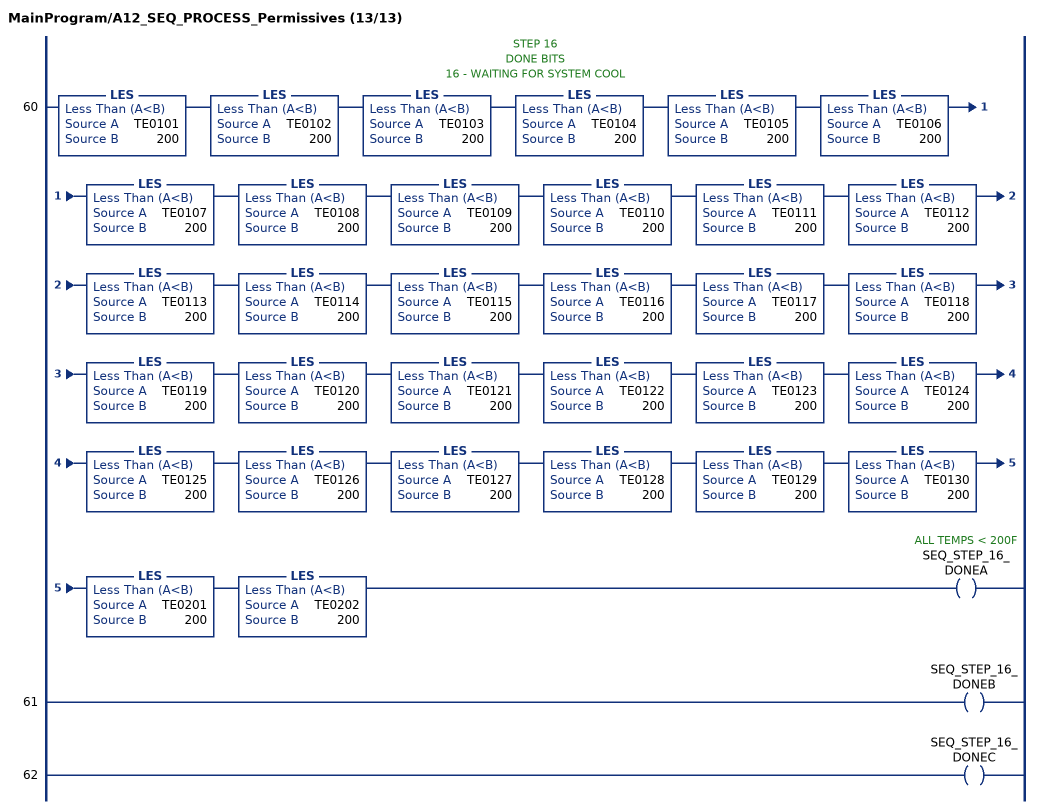
   // STEP 16
   // DONE BITS
   // 16 - WAITING FOR SYSTEM COOL
   60: LES(TE0101,200)LES(TE0102,200)LES(TE0103,200)LES(TE0104,200)LES(TE0105,200)LES(TE0106,200)LES(TE0107,200)LES(TE0108,200)LES(TE0109,200)LES(TE0110,200)LES(TE0111,200)LES(TE0112,200)LES(TE0113,200)LES(TE0114,200)LES(TE0115,200)LES(TE0116,200)LES(TE0117,200)LES(TE0118,200)LES(TE0119,200)LES(TE0120,200)LES(TE0121,200)LES(TE0122,200)LES(TE0123,200)LES(TE0124,200)LES(TE0125,200)LES(TE0126,200)LES(TE0127,200)LES(TE0128,200)LES(TE0129,200)LES(TE0130,200)LES(TE0201,200)LES(TE0202,200)OTE(SEQ_STEP_16_DONEA);
   61: OTE(SEQ_STEP_16_DONEB);
   62: OTE(SEQ_STEP_16_DONEC);
END_ROUTINE
